(* IEC 61131-3 sources: rep_b/Projects/banana_rep_st/Strategy/Task-Main, 5 files *)

(* ---- Constants.st ---- *)
VAR_GLOBAL CONSTANT

{REGION Модели контроллеров}
	PCO_5_PLUS_EXTRA_LARGE_N_O:UINT:=13;
	PCO_5_PLUS_LARGE:UINT:=10;
	PCO_5_PLUS_MEDIUM:UINT:=11;
	PCO_5_PLUS_SMALL:UINT:=12;

	PCO_5_EXTRA_LARGE_N_O:UINT:=13;
	PCO_5_EXTRA_LARGE_N_C:UINT:=17;
	PCO_5_LARGE:UINT:=10;
	PCO_5_MEDIUM:UINT:=11;
	PCO_5_SMALL:UINT:=12;
{ENDREGION}

{REGION I/O Контроллеров}
	PCO_5_PLUS_EXTRA_LARGE_N_O_UI:UINT:=8;
	PCO_5_PLUS_EXTRA_LARGE_N_O_DI:UINT:=14;
	PCO_5_PLUS_EXTRA_LARGE_N_O_AO:UINT:=4;
	PCO_5_PLUS_EXTRA_LARGE_N_O_DO:UINT:=29;

	PCO_5_PLUS_LARGE_N_O_UI:UINT:=10;
	PCO_5_PLUS_LARGE_N_O_DI:UINT:=18;
	PCO_5_PLUS_LARGE_N_O_AO:UINT:=6;
	PCO_5_PLUS_LARGE_N_O_DO:UINT:=18;

	PCO_5_PLUS_MEDIUM_N_O_UI:UINT:=8;
	PCO_5_PLUS_MEDIUM_N_O_DI:UINT:=14;
	PCO_5_PLUS_MEDIUM_N_O_AO:UINT:=4;
	PCO_5_PLUS_MEDIUM_N_O_DO:UINT:=13;

	PCO_5_PLUS_SMALL_N_O_UI:UINT:=5;
	PCO_5_PLUS_SMALL_N_O_DI:UINT:=8;
	PCO_5_PLUS_SMALL_N_O_AO:UINT:=4;
	PCO_5_PLUS_SMALL_N_O_DO:UINT:=8;

//*************************************//

    PCO_5_EXTRA_LARGE_N_O_AI:UINT:=8;
	PCO_5_EXTRA_LARGE_N_O_DI:UINT:=14;
	PCO_5_EXTRA_LARGE_N_O_AO:UINT:=4;
	PCO_5_EXTRA_LARGE_N_O_DO:UINT:=29;

	PCO_5_LARGE_N_O_AI:UINT:=10;
	PCO_5_LARGE_N_O_DI:UINT:=18;
	PCO_5_LARGE_N_O_AO:UINT:=6;
	PCO_5_LARGE_N_O_DO:UINT:=18;

	PCO_5_MEDIUM_N_O_AI:UINT:=8;
	PCO_5_MEDIUM_N_O_DI:UINT:=14;
	PCO_5_MEDIUM_N_O_AO:UINT:=4;
	PCO_5_MEDIUM_N_O_DO:UINT:=13;

	PCO_5_SMALL_N_O_AI:UINT:=5;
	PCO_5_SMALL_N_O_DI:UINT:=8;
	PCO_5_SMALL_N_O_AO:UINT:=4;
	PCO_5_SMALL_N_O_DO:UINT:=8;
{ENDREGION}

END_VAR

(* ---- GlobalVars.st ---- *)
VAR_GLOBAL

	TOT_AIN_Q:INT;
	TOT_DIN_Q:INT;
	TOT_AO_Q:INT;
	TOT_DO_Q:INT;

	start:INT;
END_VAR

(* ---- RetainGlobalVars.st ---- *)
VAR_GLOBAL RETAIN

	MasterPCOtype:UINT; //тип ведущего контроллера
	SlavePCOtype:UINT;  //тип ведомого контроллера

	Q_AI_M:INT;         //количество аналоговых входов [Master]
	Q_DI_M:INT;         //количество цифровых входов [Master]
	Q_AO_M:INT;         //количество аналоговых выходов [Master]
	Q_DO_M:INT;         //количество цифровых выходов [Master]

	Q_AI_S:INT;         //количество аналоговых входов [Slave]
	Q_DI_S:INT;         //количество цифровых входов [Slave]
	Q_AO_S:INT;         //количество аналоговых выходов [Slave]
	Q_DO_S:INT;         //количество цифровых выходов [Slave]

END_VAR

(* ---- SensorGetData.st ---- *)
(**Считывание значения входа,
  Преобразование активных входов в значения единиц измерения
  @inputNum Номер входа
  @sensorType Тип датчика
  @isPresent Существует ли вход физически
  @lowValue Нижний диапазон датчика
  @highValue Верхний диапазон датчика
  *)

FUNCTION Get_Sensor_Data:INT

VAR_INPUT
	inputNum:INT;
	sensorType:INT;
	isPresent:BOOL;
	lowValue:INT;
	highValue:INT;
END_VAR
	;
END_FUNCTION

(* ---- Main.st ---- *)
PROGRAM main

VAR
	start1:INT:=1;
END_VAR

{REGION Inizialization}

(*if X_START_SCREEN_CONFIRM == 1 then skip start page*)
X_START_SCREEN_CONFIRM:=START_SCREEN_CONFIRM;

(*Get Board type of Master controller*)
IF INIZIALIZATION_1 = FALSE THEN
	MasterPCOtype:=GET_BOARD_TYPE();    //write to Retain memory!!!
	INIZIALIZATION_1:=TRUE;
	RETURN;
END_IF;

(*Waiting user confirm plan configuration*)
IF START_SCREEN_CONFIRM = FALSE THEN
	RETURN;
END_IF;

(*Get Board type of Slave controller*)
IF INIZIALIZATION_2 = FALSE AND START_SCREEN_CONFIRM = TRUE THEN
	SlavePCOtype:=INT_TO_UINT(PLAN_GET_BOARD_TYPE);  //write to Retain memory!!!
	INIZIALIZATION_2:=TRUE;
	RETURN;
END_IF;

(*Get quantity of I/O of Master controller*)
IF INIZIALIZATION_3 = FALSE THEN

	IF MasterPCOtype = (PCO_5_PLUS_SMALL OR PCO_5_SMALL) THEN
		Q_AI_M:=PCO_5_SMALL_N_O_AI;
		Q_DI_M:=PCO_5_SMALL_N_O_DI;
		Q_AO_M:=PCO_5_SMALL_N_O_AO;
		Q_DO_M:=PCO_5_SMALL_N_O_DO;

	ELSIF MasterPCOtype = (PCO_5_PLUS_MEDIUM OR PCO_5_MEDIUM) THEN
		Q_AI_M:=PCO_5_MEDIUM_N_O_AI;
		Q_DI_M:=PCO_5_MEDIUM_N_O_DI;
		Q_AO_M:=PCO_5_MEDIUM_N_O_AO;
		Q_DO_M:=PCO_5_MEDIUM_N_O_DO;

	ELSIF MasterPCOtype = (PCO_5_PLUS_LARGE OR PCO_5_LARGE) THEN
		Q_AI_M:=PCO_5_LARGE_N_O_AI;
		Q_DI_M:=PCO_5_LARGE_N_O_DI;
		Q_AO_M:=PCO_5_LARGE_N_O_AO;
		Q_DO_M:=PCO_5_LARGE_N_O_DO;

	ELSIF MasterPCOtype = (PCO_5_PLUS_EXTRA_LARGE_N_O OR PCO_5_EXTRA_LARGE_N_O) THEN
		Q_AI_M:=PCO_5_EXTRA_LARGE_N_O_AI;
		Q_DI_M:=PCO_5_EXTRA_LARGE_N_O_DI;
		Q_AO_M:=PCO_5_EXTRA_LARGE_N_O_AO;
		Q_DO_M:=PCO_5_EXTRA_LARGE_N_O_DO;
	END_IF;

	INIZIALIZATION_3:=TRUE;

	RETURN;

END_IF;

(*Get quantity of I/O of Slave controller*)
IF INIZIALIZATION_4 = FALSE THEN

	IF SlavePCOtype = (PCO_5_PLUS_SMALL OR PCO_5_SMALL) THEN
		Q_AI_S:=PCO_5_SMALL_N_O_AI;
		Q_DI_S:=PCO_5_SMALL_N_O_DI;
		Q_AO_S:=PCO_5_SMALL_N_O_AO;
		Q_DO_S:=PCO_5_SMALL_N_O_DO;

	ELSIF SlavePCOtype = (PCO_5_PLUS_MEDIUM OR PCO_5_MEDIUM) THEN
		Q_AI_S:=PCO_5_MEDIUM_N_O_AI;
		Q_DI_S:=PCO_5_MEDIUM_N_O_DI;
		Q_AO_S:=PCO_5_MEDIUM_N_O_AO;
		Q_DO_S:=PCO_5_MEDIUM_N_O_DO;

	ELSIF SlavePCOtype = (PCO_5_PLUS_LARGE OR PCO_5_LARGE) THEN
		Q_AI_S:=PCO_5_LARGE_N_O_AI;
		Q_DI_S:=PCO_5_LARGE_N_O_DI;
		Q_AO_S:=PCO_5_LARGE_N_O_AO;
		Q_DO_S:=PCO_5_LARGE_N_O_DO;

	ELSIF SlavePCOtype = (PCO_5_PLUS_EXTRA_LARGE_N_O OR PCO_5_EXTRA_LARGE_N_O) THEN
		Q_AI_S:=PCO_5_EXTRA_LARGE_N_O_AI;
		Q_DI_S:=PCO_5_EXTRA_LARGE_N_O_DI;
		Q_AO_S:=PCO_5_EXTRA_LARGE_N_O_AO;
		Q_DO_S:=PCO_5_EXTRA_LARGE_N_O_DO;
	END_IF;

	INIZIALIZATION_4:=TRUE;

	RETURN;

END_IF;

TOT_AIN_Q:= Q_AI_M + Q_AI_S;
TOT_DIN_Q:= Q_DI_M + Q_DI_S;
TOT_AO_Q:= Q_AO_M + Q_AO_S;
TOT_DO_Q:= Q_DO_M + Q_DO_S;

{ENDREGION}

{REGION AIN SCREEN CONFIG INIZIALIZATION}

IF (INIZIALIZATION_5 = FALSE) THEN
	IF PCO_QUANTITY = 1 THEN
		AIN_MASTER_FLAG_B_6:= Q_AI_M > 5;
		AIN_MASTER_FLAG_B_7:= Q_AI_M > 5;
		AIN_MASTER_FLAG_B_8:= Q_AI_M > 5;
		AIN_MASTER_FLAG_B_9:= Q_AI_M > 8;
		AIN_MASTER_FLAG_B_10:= Q_AI_M > 8;

		AIN_SLAVE_FLAG_B_1:= FALSE;
		AIN_SLAVE_FLAG_B_2:= FALSE;
		AIN_SLAVE_FLAG_B_3:= FALSE;
		AIN_SLAVE_FLAG_B_4:= FALSE;
		AIN_SLAVE_FLAG_B_5:= FALSE;
		AIN_SLAVE_FLAG_B_6:= FALSE;
		AIN_SLAVE_FLAG_B_7:= FALSE;
		AIN_SLAVE_FLAG_B_8:= FALSE;
		AIN_SLAVE_FLAG_B_9:= FALSE;
		AIN_SLAVE_FLAG_B_10:= FALSE;
	END_IF;

	IF PCO_QUANTITY = 2 THEN
		AIN_MASTER_FLAG_B_6:= Q_AI_M > 5;
		AIN_MASTER_FLAG_B_7:= Q_AI_M > 5;
		AIN_MASTER_FLAG_B_8:= Q_AI_M > 5;
		AIN_MASTER_FLAG_B_9:= Q_AI_M > 8;
		AIN_MASTER_FLAG_B_10:= Q_AI_M > 8;

		AIN_SLAVE_FLAG_B_1:= TRUE;
		AIN_SLAVE_FLAG_B_2:= TRUE;
		AIN_SLAVE_FLAG_B_3:= TRUE;
		AIN_SLAVE_FLAG_B_4:= TRUE;
		AIN_SLAVE_FLAG_B_5:= TRUE;
		AIN_SLAVE_FLAG_B_6:= Q_AI_M > 5;
		AIN_SLAVE_FLAG_B_7:= Q_AI_M > 5;
		AIN_SLAVE_FLAG_B_8:= Q_AI_M > 5;
		AIN_SLAVE_FLAG_B_9:= Q_AI_M > 8;
		AIN_SLAVE_FLAG_B_10:= Q_AI_M > 8;
	END_IF;

INIZIALIZATION_5:=TRUE;
END_IF;

{ENDREGION}

start:=Get_Sensor_Data(5,ST_B_1,AIN_MASTER_FLAG_B_1,0,0);

END_PROGRAM
